FUNCTION_BLOCK HMI_BUTTONS (* Human machine interface for input *)
  (* Standard: 61499-2 *)
  (* Version 0.1, 2002-01-08, JHC, Rockwell Automation, Added DLY FB as example. *)
  (* Version 0.0, 2000-05-27, JHC, Rockwell Automation *)
  (* Compiler header: package fb.rt.festo1;import fb.rt.hmi.*; *)
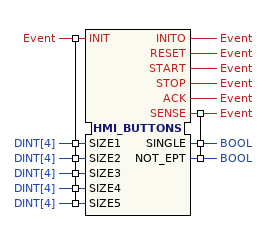
  EVENT_INPUT
    INIT WITH SIZE1, SIZE2, SIZE3, SIZE4, SIZE5; (* Initialization Request *)
  END_EVENT
  EVENT_OUTPUT
    INITO; (* Initialization Confirm *)
    RESET; (* Execution Confirmation *)
    START; (* Execution Confirmation *)
    STOP; (* Execution Confirmation *)
    ACK; (* Execution Confirmation *)
    SENSE WITH SINGLE, NOT_EPT; (* Execution Confirmation *)
  END_EVENT
  VAR_INPUT
    SIZE1 : ARRAY [0..3] OF DINT;
    SIZE2 : ARRAY [0..3] OF DINT;
    SIZE3 : ARRAY [0..3] OF DINT;
    SIZE4 : ARRAY [0..3] OF DINT;
    SIZE5 : ARRAY [0..3] OF DINT;
  END_VAR
  VAR_OUTPUT
    SINGLE : BOOL; (* Output event qualifier *)
    NOT_EPT : BOOL; (* Output event qualifier *)
  END_VAR
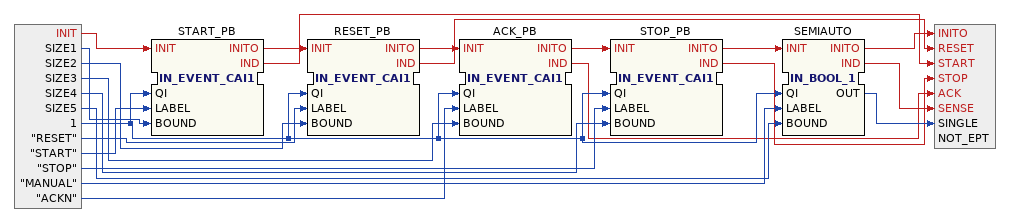
  FBS
    START_PB : IN_EVENT_CAI1;
    RESET_PB : IN_EVENT_CAI1;
    STOP_PB : IN_EVENT_CAI1;
    ACK_PB : IN_EVENT_CAI1;
    SEMIAUTO : IN_BOOL_1;
  END_FBS
  EVENT_CONNECTIONS
    INIT TO START_PB.INIT;
    START_PB.INITO TO RESET_PB.INIT;
    RESET_PB.INITO TO ACK_PB.INIT;
    ACK_PB.INITO TO STOP_PB.INIT;
    STOP_PB.INITO TO SEMIAUTO.INIT;
    SEMIAUTO.INITO TO INITO;
    RESET_PB.IND TO RESET;
    START_PB.IND TO START;
    STOP_PB.IND TO STOP;
    ACK_PB.IND TO ACK;
    SEMIAUTO.IND TO SENSE;
  END_CONNECTIONS
  DATA_CONNECTIONS
    1 TO RESET_PB.QI;
    1 TO START_PB.QI;
    1 TO STOP_PB.QI;
    1 TO ACK_PB.QI;
    1 TO SEMIAUTO.QI;
    "RESET" TO RESET_PB.LABEL;
    "START" TO START_PB.LABEL;
    "STOP" TO STOP_PB.LABEL;
    "MANUAL" TO SEMIAUTO.LABEL;
    "ACKN" TO ACK_PB.LABEL;
    SEMIAUTO.OUT TO SINGLE;
    SIZE1 TO START_PB.BOUND;
    SIZE2 TO RESET_PB.BOUND;
    SIZE3 TO ACK_PB.BOUND;
    SIZE4 TO STOP_PB.BOUND;
    SIZE5 TO SEMIAUTO.BOUND;
  END_CONNECTIONS
END_FUNCTION_BLOCK
